INTERFACE I_HE_SATT_PhotonEnergy_eV


PROPERTY Error : BOOL
GET
END_GET
END_PROPERTY


PROPERTY Value : LREAL
GET
END_GET
END_PROPERTY

END_INTERFACE

(* stored: Version 1.1.0.1
   Itf I_HE_SATT_PhotonEnergy_eV: Id {39eb1a50-4543-4e7c-b134-b201f0fac44d}
   Property Error: Id {6b232ec1-7d71-45b4-9246-0c91ab1bd468}
   Get Get: Id {6d56e98b-9a26-40b5-af0c-6bad7fbda8d7}
   Property Value: Id {a6e11785-360b-4b75-99f3-3cdf7544e171}
   Get Get: Id {1ce52de1-5625-40e3-8d42-8448fd7286de} *)
